Fanuc KAREL source: kt00477.KL

-- PROVISIONAL review KL for V1013-1; original PC SHA256 a3cc8cc4d89afce374338aaf0a18ecf9bf3231d564fcdafc6156e0cf166f01ef
-- Incomplete behavior may be omitted. Consult companion uncertainty JSON. Do not deploy.
PROGRAM KT00477
%NOLOCKGROUP
-- UNRESOLVED_DECL P1 type=000101
-- UNRESOLVED_DECL P2 type=000101
-- UNRESOLVED_DECL OUT type=000199
BEGIN
  -- UNRESOLVED_PC offsets 5-34; opcodes 49,49,60,7E,4A
  -- UNRESOLVED_PC offsets 39-43; opcodes 7F
END KT00477
